PROGRAM PRG_SystemInfo
VAR
	bSystemInfoLoaded : BOOL := FALSE;
END_VAR

IF NOT bSystemInfoLoaded THEN
	
	GVL_HMI.stInfo.sApplication := 'Automated Sample Recovery System';
	GVL_HMI.stInfo.sProjectId := 'TE 1063';
	GVL_HMI.stInfo.sTwincatVersion := 'v3.1 4024.5, Runtime v3.1.4024.53';
	GVL_HMI.stInfo.sVSVersion := 'VS 2017 Shell v15.0.35116.124 D15.9';
	GVL_HMI.stInfo.rSoftwareVersion := 0.0;
	GVL_HMI.stInfo.sDate := 'December 2025';
	
	bSystemInfoLoaded := TRUE;
END_IF

END_PROGRAM

(* stored: Version 1.1.0.1, ProductVersion 3.1.4024.15
   POU PRG_SystemInfo: Id {3ecda4e7-3da9-4b19-a635-328f489eb573}, SpecialFunc None *)
